(* IEC 61131-3 sources: SRCI/RobotLibrary/RobotLibrary/POUs/Trigger/MC_SetTriggerRegister, 1 file *)

(* ---- MC_SetTriggerRegisterFB.st ---- *)
/// Trigger "Actions" based on I/O related events (e.g. change of DI’s state)
FUNCTION_BLOCK MC_SetTriggerRegisterFB EXTENDS RobotLibraryBaseExecuteFB
// -------------------------------------------------------------------------
//  SRCI Robot Library
// -------------------------------------------------------------------------
//
//  Object:      SetTriggerRegisterFB
//  Author:      Thorsten Brach
//  Date:        2024-06-01
//
//  Description:
//
//
//  Copyright:
//    (C) 2024 Thorsten Brach. All rights reserved
//             Licensed under the LGPL-3.0 license.
//
//  Disclaimer:
//    This project is provided without any guarantee and can be used for
//    private and commercial purposes. Any use is at the user’s
//    own risk and responsibility.
//
// -------------------------------------------------------------------------
VAR_INPUT
  /// Processing mode
  ProcessingMode   : ProcessingMode;
  /// command parameter
  ParCmd           : SetTriggerRegisterParCmd;
END_VAR
VAR_OUTPUT
  /// Command is transferred and confirmed by the RC
  CommandBuffered  : BOOL;
  /// TRUE, when the monitoring of the input parameter values is active.
  MonitoringActive : BOOL;
  /// command results
  OutCmd           : SetTriggerRegisterOutCmd;
END_VAR

VAR
  /// internal copy of command parameter
 _parCmd           : SetTriggerRegisterParCmd;
  /// command data to send
 _command          : SetTriggerRegisterSendData;
  /// response data received
 _response         : SetTriggerRegisterRecvData;
END_VAR

  SUPER^(AxesGroup := AxesGroup);

END_FUNCTION_BLOCK

METHOD CheckParameterChanged : BOOL
VAR_IN_OUT
  /// Robot assignment of function
  AxesGroup    : AxesGroup;
END_VAR

  // Check ParCmd Size is > 0, becaue MemCmp does not work correctly with size = 0
  IF (SIZEOF(ParCmd) = 0)
  THEN
    RETURN;
  END_IF

  // compare memory
  CheckParameterChanged := ( MemCmp(ADR(ParCmd), ADR(_parCmd), SIZEOF(ParCmd)) <> RobotLibraryConstants.OK );

  IF ( CheckParameterChanged )
  THEN
    // update internal copy of parameters
   _parCmd := ParCmd;
    // inc parameter sequence
   _command.ParSeq := _command.ParSeq + 1;
    // update command data
    CommandData := CreateCommandPayload(); // ( Access via reference to rCommandFB in ACR )
    // notify active command register
    AxesGroup.Acyclic.ActiveCommandRegister.NotifyParameterChanged := _uniqueID;
  END_IF

END_METHOD

METHOD INTERNAL CreateCommandPayload : SendData
// Table 6-579: Sent CMD payload (PLC to RC) of "SetTriggerRegister"
// --------------------------
// Header
// --------------------------
// Byte 00 : UINT  - Type HB
// Byte 01 :       - Type LB
// Byte 02 : USINT - Reserve | ExecutionMode
// Byte 03 : USINT - ParSeq  | Priority
// --------------------------
// Datablock
// --------------------------
// Byte 04 : SINT  EmitterID[0];
// Byte 05 : SINT  EmitterID[1];
// Byte 06 : SINT  EmitterID[2];
// Byte 07 : SINT  EmitterID[3];
// Byte 08 : SINT  ListenerID;
// Byte 09 : BYTE  Reserved;
// Byte 10 : INT   IntValue_1;
// Byte 11 :       IntValue_1;
// Byte 12 : INT   IntValue_2;
// Byte 13 :       IntValue_2;
// Byte 14 : REAL  RealValue_1;
// Byte 15 :       RealValue_1;
// Byte 16 :       RealValue_1;
// Byte 17 :       RealValue_1;
// Byte 18 : REAL  RealValue_2;
// Byte 19 :       RealValue_2;
// Byte 20 :       RealValue_2;
// Byte 21 :       RealValue_2;
// Byte 22 : SINT  TriggerMode;
// Byte 23 : USINT Index;
// Byte 24 : USINT BitIndex;

  // set command parameter
  _command.CmdTyp       :=  CmdType.SetTriggerRegister;
  _command.ExecMode     :=  ExecMode;
  _command.ParSeq       := _command.ParSeq;
  _command.Priority     :=  Priority;

  _command.EmitterID[0] := _parCmd.EmitterID;
  _command.EmitterID[1] := 0;
  _command.EmitterID[2] := 0;
  _command.EmitterID[3] := 0;
  _command.ListenerID   := _parCmd.ListenerID;
  _command.Reserve      := 0;
  _command.IntValue     := _parCmd.IntValue;
  _command.RealValue    := _parCmd.RealValue;
  _command.TriggerMode  := _parCmd.TriggerMode;
  _command.Index        := _parCmd.Index;
  _command.BitIndex     := _parCmd.BitIndex;

  // copy command data to header
  _cmdHeader := _command;
  // call base implementation to copy header to payload buffer
  CreateCommandPayload := SUPER^.CreateCommandPayload();

  // add command.EmitterID[0]
  CreateCommandPayload.AddSint(_command.EmitterID[0]);
  // add command.EmitterID[1]
  CreateCommandPayload.AddSint(_command.EmitterID[1]);
  // add command.EmitterID[2]
  CreateCommandPayload.AddSint(_command.EmitterID[2]);
  // add command.EmitterID[3]
  CreateCommandPayload.AddSint(_command.EmitterID[3]);
  // add command.ListenerID
  CreateCommandPayload.AddSint(_command.ListenerID);
  // add command.Reserve
  CreateCommandPayload.AddByte(_command.Reserve);
  // add command.IntValue[1]
  CreateCommandPayload.AddInt(_command.IntValue[1]);
  // add command.IntValue[2]
  CreateCommandPayload.AddInt(_command.IntValue[2]);
  // add command.RealValue[1]
  CreateCommandPayload.AddReal(_command.RealValue[1]);
  // add command.RealValue[2]
  CreateCommandPayload.AddReal(_command.RealValue[2]);
  // add command.TriggerMode
  CreateCommandPayload.AddSint(_command.TriggerMode);
  // add command.Index
  CreateCommandPayload.AddUsint(_command.Index);
  // add command.BitIndex
  CreateCommandPayload.AddUsint(_command.BitIndex);

END_METHOD

METHOD FB_init : BOOL
VAR_INPUT
  /// if TRUE, the retain variables are initialized (warm start / cold start)
	bInitRetains : BOOL;
  /// if TRUE, the instance afterwards gets moved into the copy code (online change)
	bInCopyCode  : BOOL;
END_VAR

  MyType := 'MC_SetTriggerRegisterFB';

  ExecMode := ExecutionMode.PARALLEL;

END_METHOD

METHOD PROTECTED OnCall
VAR_IN_OUT
  /// Robot assignment of function
  AxesGroup : AxesGroup;
END_VAR

  // call base implementation
  SUPER^.OnCall(AxesGroup := AxesGroup);

  CASE _stepCmd OF

    00:  IF ( _execute_R.Q )
         THEN
           // set busy flag
           Busy := TRUE;
           // Reset command outputs
           MemSet(ADR(OutCmd),0,SIZEOF(OutCmd));
           // apply command parameter
          _parCmd := ParCmd;
           // init parameter sequence
          _command.ParSeq := 1;
           // set timeout
           SetTimeout(PT := _timeoutCmd, rTimer := _timerCmd);
           // inc step counter
          _stepCmd := _stepCmd + 1;
  	     END_IF

    01:  // create command data
         CommandData := CreateCommandPayload();
         // Add command to active command register
        _uniqueID := AxesGroup.Acyclic.ActiveCommandRegister.AddCmd( pCommandFB := ADR(THIS^ ));
         // set timeout
         SetTimeout(PT := _timeoutCmd, rTimer := _timerCmd);
         // inc step counter
        _stepCmd := _stepCmd + 1;

    02:  // Wait for responce received
         IF ( _responseReceived )
         THEN
           // reset response received flag
          _responseReceived := FALSE;
           // reset MonitoringActive flag
           MonitoringActive := FALSE;

           CASE  _response.State
           OF
             CmdMessageState.BUFFERED : CommandBuffered  := TRUE;
             CmdMessageState.ACTIVE   : MonitoringActive := TRUE;
             CmdMessageState.DONE     : Done             := TRUE;
             CmdMessageState.ERROR    : Error            := TRUE;
  				 END_CASE

           // Done, Aborted or Error ?
           IF (_response.State >= CmdMessageState.DONE )
           THEN
             // Reset Busy flag
             Busy := FALSE;
             // Update results
             OutCmd.InvocationCounter := _response.InvocationCounter;
             OutCmd.OriginID          := _response.OriginID;
             // set timeout
             SetTimeout(PT := _timeoutCmd, rTimer := _timerCmd);
             // inc step counter
            _stepCmd := _stepCmd + 1;
  				 END_IF
         END_IF

    03: IF ( NOT Execute)
        THEN
          Reset();
  			END_IF
  ELSE
    // invalid step
    ErrorID := RobotLibraryEvents.ERR_INVALID_STEP;
  END_CASE

  // Cancel
  IF (Busy) AND (NOT Execute)
  THEN
    // try to remove cmd
    AxesGroup.Acyclic.ActiveCommandRegister.RemoveCmd(_uniqueID);
  END_IF

  // Reset FB
  IF ( NOT Execute )
  THEN
    Reset();
  END_IF

END_METHOD

METHOD INTERNAL ParseResponsePayload : DINT
// Table 6-580: Received CMD payload (RC to PLC) of "SetTriggerRegister"
// --------------------------
// Header
// --------------------------
// Byte 00 : USINT   - ParSeq | State
// Byte 01 : SINT    - AlarmMessageSeverity
// Byte 02 : UINT    - AlarmMessageCode HB
// Byte 03 :         - AlarmMessageCode LB
// --------------------------
// Datablock
// --------------------------
// Byte 04 : USINT   - InvocationCounter
// Byte 05 : SINT    - Reserve
// Byte 06 : INT     - OriginID LW HB
// Byte 07 :         - OriginID LW LB
VAR_INPUT
  /// Response data
  ResponseData : RecvData;
END_VAR

  // call base implementation to parse the header from payload buffer
  ResponseData.PayloadPtr := SUPER^.ParseResponsePayload(ResponseData);

  // copy parsed header to response
  _response.ParSeq               := _rspHeader.ParSeq;
  _response.State                := _rspHeader.State;
  _response.AlarmMessageSeverity := _rspHeader.AlarmMessageSeverity;
  _response.AlarmMessageCode     := _rspHeader.AlarmMessageCode;

  // Get Response.InvocationCounter
  _response.InvocationCounter := ResponseData.GetUsint();
  // Get Response.Reserve
  _response.Reserve := ResponseData.GetSint();
  // Get Response.OriginID
  _response.OriginID := ResponseData.GetInt();

END_METHOD

METHOD PROTECTED Reset : DINT
VAR_INPUT
END_VAR

  Reset := SUPER^.Reset();

  Done             := FALSE;
  Busy             := FALSE;
  MonitoringActive := FALSE;
  CommandBuffered  := FALSE;

END_METHOD
